FUNCTION_BLOCK INTERNAL FlagListExtender
VAR
	_iList		: I_FlagList;
END_VAR

PROPERTY INTERNAL List : I_FlagList
GET
List := _iList;
END_GET
SET
_iList := List;
END_SET
END_PROPERTY

END_FUNCTION_BLOCK

(* stored: Version 1.1.0.1
   POU FlagListExtender: Id {ec7afdb6-076b-4e9c-8d6c-36629837f2f3}, SpecialFunc None
   Property List: Id {aa5b4145-1ceb-48c4-9a9d-987d7cd30beb}
   Get Get: Id {869770d4-278b-41af-87df-03ff9d205269}
   Set Set: Id {a3893ab2-b7d5-4e86-8d6c-c3dfec6f9578} *)
